PROGRAM EtherCatDiagnosis
VAR
	fb_GetLocalAmsNetId		: FB_GetLocalAmsNetId;
	fb_getConfiguredSlaves 	: FB_EcGetConfSlaves;
	fb_getScannedSlaves 	: FB_EcGetScannedSlaves; 
	fb_GetLicenses 			: FB_GetLicenses;		
	fb_CpuUsage				: TC_CpuUsage;
	
	pArrConfiguredSlaveData : POINTER TO ARRAY[0..EC_MAX_SLAVES] OF ST_EcSlaveConfigData;
	pArrScannedSlaveData  	: POINTER TO ARRAY[0..EC_MAX_SLAVES] OF ST_EcSlaveScannedData;
	
	fb_plcSymbolInfo : PLC_ReadSymInfoByName;

END_VAR

fb_GetLocalAmsNetId(
	bExecute 			:= ,
	tTimeOut 			:= ,
	bBusy 				=> ,
	bError				=> ,
	nErrId 				=> ,
	AddrString 			=> ,
	AddrBytes 			=> );

fb_getConfiguredSlaves(
	sNetId				:= fb_GetLocalAmsNetId.AddrString,
	pArrEcConfSlaveInfo	:= pArrConfiguredSlaveData,
	cbBufLen 			:= SIZEOF(pArrConfiguredSlaveData),
	bExecute 			:= ,
	tTimeout 			:= ,
	bBusy 				=> ,
	bError 				=> ,
	nErrorId 			=> ,
	nSlaves 			=> );
	
fb_getScannedSlaves(
	bExecute 				:= ,
	sNetId 					:= ,
	pArrEcScannedSlaveInfo 	:= pArrScannedSlaveData,
	cbBufLen 				:= SIZEOF(pArrScannedSlaveData),
	tTimeout 				:= ,
	bBusy 					=> ,
	bError 					=> ,
	nErrorId 				=> ,
	nSlaves 				=> );

fb_GetLicenses(
	bExecute 			:= ,
	tTimeout 			:= ,
	sNetId 				:= ,
	bBusy 				=> ,
	bError 				=> ,
	nErrorId 			=> ,
	nValidLicenses 		=>,
	aValidLicenses 		=> ,
	nInvalidLicenses 	=>,
	aInvalidLicenses 	=> );
	
fb_CpuUsage(
	NETID := ,
	START := ,
	TMOUT := ,
	BUSY => ,
	ERR => ,
	ERRID => ,
	USAGE => );
	
fb_plcSymbolInfo(
	NETID :=,
	PORT :=,
	SYMNAME :=,
	START:=,
	TMOUT :=,
	BUSY =>,
	ERR =>,
	ERRID=>,
	SYMINFO =>);

END_PROGRAM

(* stored: Version 1.1.0.1, ProductVersion 3.1.4024.12
   POU EtherCatDiagnosis: Id {6e4fc343-10cc-41c2-9849-69fd2ebb5434}, SpecialFunc None *)
